FUNCTION_BLOCK GF_Befuellen	EXTENDS FB_Basis
VAR_INPUT
	// Instanzieren von Sensoren mit Interfaces
	I_Level		:I_Sensor;
	// Instanzieren von Aktoren mit Interfaces
	I_Ventil	:I_Magnetventil;
	// Rezeptparameter durch Controlword
	I_CW		:RezeptControlWord;	
END_VAR
VAR_OUTPUT
	O_SW		:RezeptStatusWord;
END_VAR
VAR
	
END_VAR

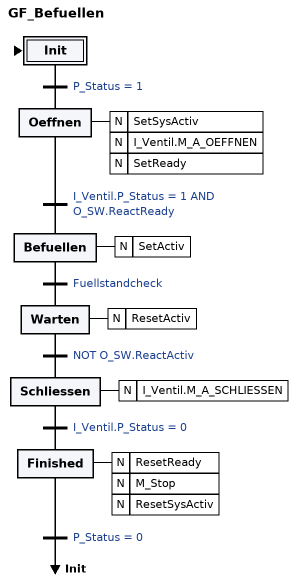
INITIAL_STEP Init:
END_STEP
TRANSITION FROM Init TO Oeffnen
    := P_Status = 1;
END_TRANSITION
STEP Oeffnen:
    SetSysActiv(N);
    I_Ventil.M_A_OEFFNEN(N);
    SetReady(N);
END_STEP
TRANSITION FROM Oeffnen TO Befuellen
    := I_Ventil.P_Status = 1 AND O_SW.ReactReady;
END_TRANSITION
STEP Befuellen:
    SetActiv(N);
END_STEP
TRANSITION FROM Befuellen TO Warten
    := Fuellstandcheck;
END_TRANSITION
STEP Warten:
    ResetActiv(N);
END_STEP
TRANSITION FROM Warten TO Schliessen
    := NOT O_SW.ReactActiv;
END_TRANSITION
STEP Schliessen:
    I_Ventil.M_A_SCHLIESSEN(N);
END_STEP
TRANSITION FROM Schliessen TO Finished_
    := I_Ventil.P_Status = 0;
END_TRANSITION
STEP Finished_:  // name as stored: Finished 
    ResetReady(N);
    M_Stop(N);
    ResetSysActiv(N);
END_STEP
TRANSITION FROM Finished_ TO Init
    := P_Status = 0;
END_TRANSITION

TRANSITION Fuellstandcheck:
// Prüfen welche Grundfunktion verwendet wird
IF I_CW.Enlteermenge > 0 THEN
	// Bedingung
	IF  I_CW.Enlteermenge < I_Level.P_Messwert THEN
		Fuellstandcheck := TRUE;
		
	ELSE 
		Fuellstandcheck := FALSE;
	END_IF
END_IF

// Prüfen welche Grundfunktion verwendet wird
IF I_CW.Pumpmenge > 0 THEN
	// Bedingung
	IF  I_CW.Pumpmenge < I_Level.P_Messwert THEN
		Fuellstandcheck := TRUE;
	ELSE 
		Fuellstandcheck := FALSE;
	END_IF
END_IF
END_TRANSITION

ACTION ResetActiv:
O_SW.ReactActiv := FALSE;
O_SW.GF7Activ := FALSE;
END_ACTION

ACTION ResetReady:
O_SW.ReactReady := FALSE;
END_ACTION

ACTION ResetSysActiv:
GVL.SysState := 0;
// Für Debug
GVL.Debug_SekStart := 0;
END_ACTION

ACTION SetActiv:
O_SW.ReactActiv := TRUE;
O_SW.GF7Activ := TRUE;
END_ACTION

ACTION SetReady:
O_SW.ReactReady := TRUE;
END_ACTION

ACTION SetSysActiv:
GVL.SysState := 1;
END_ACTION

END_FUNCTION_BLOCK

(* stored: Version 1.1.0.1, ProductVersion 3.1.4024.12
   POU GF_Befuellen: Id {a2b409ce-e0b4-4790-bbb6-ecfa82d1d496}, SpecialFunc None
   Folder 01_Aktionen: Id {0d7df3fb-47f4-4495-b978-56a9f3a832e4}
   Folder 02_Transitions: Id {dda3a0c4-e8f9-4c9e-a611-30798de31893}
   Transition Fuellstandcheck: Id {34ac417c-4efe-466c-a9ee-bde5e34579b7}
   Action ResetActiv: Id {26b6df95-fd29-4c3a-9a68-95c3f69bf336}
   Action ResetReady: Id {23662753-2ca6-4c22-a1c0-77f706883224}
   Action ResetSysActiv: Id {67fdda91-07d5-47da-a0da-171955fb3e5f}
   Action SetActiv: Id {07070a43-bcc7-45f3-9381-b8da515e0b5c}
   Action SetReady: Id {89c38aa9-37eb-4727-b8e7-0908130829dd}
   Action SetSysActiv: Id {13869d2e-1a10-48e8-8d39-cb3815ca389a} *)
